// Base class of all classes in the FisoThemes Standard Library.
{attribute 'enable_dynamic_creation'}
{attribute 'reflection'}
{attribute 'no_assign'}
{attribute 'no_explicit_call' := 'direct call for this function block is not allowed'} 
FUNCTION_BLOCK FsFB_Object IMPLEMENTS FsI_Object

// Private local variable to store object's size
METHOD PRIVATE _Size : FsT_Size
VAR_INPUT
	Accessor : FsT_Accessor;
	Data : FsT_Size;
END_VAR
VAR_INST
	Store : FsT_Size;
END_VAR
CASE Accessor OF
	FsT_Accessor.Set:
		_Size := Store := Data;
	FsT_Accessor.Get:
		_Size := Store;
	END_CASE
END_METHOD

// Pointer to the object in memory.
PROPERTY FINAL Address : FsT_Ptr
GET
Address := THIS;
END_GET
END_PROPERTY

// A string that represents the type of the object if the object is created dynamically.
// Classes indeed for dynamic use must override this property.
PROPERTY PROTECTED DynamicTypeName : FsT_Str
GET
DynamicTypeName := 'FsFB_Object';
END_GET
END_PROPERTY

{attribute 'hide'}
METHOD FB_init : BOOL
VAR_INPUT
	bInitRetains : BOOL; // if TRUE, the retain variables are initialized (warm start / cold start)
	bInCopyCode : BOOL;  // if TRUE, the instance afterwards gets moved into the copy code (online change)
END_VAR
VAR
	sTypeName : FsT_Str;
	i : FsT_Size := 0;
END_VAR
// If size has already been initialised then don't run this again.
IF THIS^.Size <> 0 THEN RETURN; END_IF

CASE THIS^.MemoryArea OF
// Attempt to get size of object.
	FsT_MemArea.Static:
	// If object in static memory try and look for it using the TcCOM object server and get it's size.
		FOR i := SIZEOF(THIS^) TO FsParam_Core.INFO_SCAN_SIZE DO
			sTypeName := FsF_GetTypeNameByAddress(THIS, i);
			IF sTypeName <> '' THEN EXIT; END_IF
			END_FOR
		THIS^._Size(FsT_Accessor.Set, i);
ELSE
// In any other case just return the base object size.
	THIS^._Size(FsT_Accessor.Set, SIZEOF(THIS^));
	END_CASE
END_METHOD

// Represents the path to the object.
PROPERTY FINAL InstancePath : FsT_LStr
GET
CASE THIS^.MemoryArea OF
	FsT_MemArea.Static: 
		InstancePath := FsF_GetVariablePathByAddress(THIS, THIS^.Size);
	FsT_MemArea.Dynamic:
		InstancePath := '<Dynamic>';
	FsT_MemArea.CNC:
		InstancePath := '<Unsupported>';
ELSE
	InstancePath := '<Unknown>';
	END_CASE
END_GET
END_PROPERTY

// Checks if the current object is the same as (reference-wise) object as the input object.
METHOD FINAL Is : BOOL
VAR_INPUT
	ipObject : FsI_Object;
END_VAR
IF ipObject <> 0 THEN Is := ipObject.Address = THIS; END_IF
END_METHOD

// Memory area that the object is allocated in.
PROPERTY FINAL MemoryArea : FsT_MemArea
GET
MemoryArea := Tc2_System.F_CheckMemoryArea(THIS, 1);
END_GET
END_PROPERTY

//  Size of the object in bytes.
PROPERTY Size : FsT_Size
GET
Size := THIS^._Size(FsT_Accessor.Get, 0);
END_GET
END_PROPERTY

// Converts this object to a string representation.
METHOD ToString : FsT_LStr
ToString := THIS^.TypeName;
END_METHOD

// A string that represents the type of the object.
PROPERTY FINAL TypeName : FsT_Str
GET
CASE THIS^.MemoryArea OF
	FsT_MemArea.Static: 
		TypeName := FsF_GetTypeNameByAddress(THIS, THIS^.Size);
	FsT_MemArea.Dynamic:
		TypeName := THIS^.DynamicTypeName;
	FsT_MemArea.CNC:
		TypeName := '<Unsupported>';
ELSE
	TypeName := '<Unknown>';
	END_CASE
END_GET
END_PROPERTY

END_FUNCTION_BLOCK

(* stored: Version 1.1.0.1, ProductVersion 3.1.4024.4
   POU FsFB_Object: Id {b9a7d797-4e3c-4bd7-a9f4-98928c915162}, SpecialFunc None
   Folder Methods: Id {9e68c5d1-f194-4f3e-b6b3-7681e0f201d7}
   Folder Properties: Id {6e68efcf-a06b-4741-a90c-39cba0c68559}
   Method _Size: Id {9947d38c-b13b-4f37-bc4a-f1fd93a541f7}
   Property Address: Id {7007c1fb-a7ab-4291-aa3a-d0ddd5d42f4e}
   Get Get: Id {bd783e5b-6e26-4874-9513-4747948415c4}
   Property DynamicTypeName: Id {5d51a533-0704-4c7c-9757-7a76d7dbe92e}
   Get Get: Id {bdb32137-9214-4f98-8796-df49473f1713}
   Method FB_init: Id {5a15df2b-2053-43e1-92ac-307f29102340}
   Property InstancePath: Id {218ed01a-d849-4c65-abf6-b55439d7517f}
   Get Get: Id {0f631ee9-366e-4d13-8b5f-ec18d6b4567b}
   Method Is: Id {f68eded3-5c4f-48e4-a1f7-d41bc7feec35}
   Property MemoryArea: Id {e32d98e4-15ab-4c88-8320-1cf851d9094c}
   Get Get: Id {0cb27507-fdbf-437b-a27f-717e8f9abf9a}
   Property Size: Id {ec229d8f-c9f5-4131-ac66-6ff8ee3e8ff6}
   Get Get: Id {5c227faa-2113-4148-a339-352f5334e00b}
   Method ToString: Id {fd669478-cc29-4dd3-b596-b7591a7cd36c}
   Property TypeName: Id {798da96d-0670-4365-8189-eab7f1df96d3}
   Get Get: Id {aea9ec0c-e0a1-480b-82b8-9eff58306bd6} *)
